FUNCTION DataToIndex : UINT


VAR_INPUT

data       : POINTERTOUINT;;

dataLength : UINT;;

value      : UINT;;

    END_VAR


VAR

count : UINT;;

    END_VAR

END_FUNCTION

END_PROGRAM


FOR count := 1 TO dataLength BY 1 DO

IF data^= value THEN

DataToIndex := count;

RETURN;

        END_IF

data := data + SIZEOF (data^);

    END_FOR

END_FUNCTION

(* stored: Version 1.1.0.1, ProductVersion 3.1.4022.6
   POU DataToIndex: Id {c1d7d7e4-c94c-47fa-b620-2c1290dbaa30}, SpecialFunc None *)
